{attribute addProperty BoxType "EL5112-0000-0016"}
{attribute addProperty Id "ENC_Status_Channel_1AT %I*ENC_Status_Channel_D7AAABA7128160ENC_Control_Channel_1AT %Q*ENC_Control_Channel_C4E6260B4860WcStateAT %I*WcState_F855686C1620InfoDataAT %I*InfoData_BC63D37F80100"}
{attribute addProperty CRC "1457377746"}
{attribute addProperty SizeInBites "272"}
{attribute addProperty SizeInBytes "34"}
TYPE EL5112_0DC93E84 :
STRUCT
	{attribute addProperty Name "ENC_Status_Channel_1"}
	ENC_Status_Channel_1 : ENC_Status_Channel_D7AAABA7;
	{attribute addProperty Name "ENC_Control_Channel_1"}
	ENC_Control_Channel_1 : ENC_Control_Channel_C4E6260B;
	{attribute addProperty Name "WcState"}
	WcState : WcState_F855686C;
	{attribute addProperty Name "InfoData"}
	InfoData : InfoData_BC63D37F;
END_STRUCT
END_TYPE

(* stored: Version 1.2.0.0, ProductVersion 3.1.4024.9
   DUT EL5112_0DC93E84: Id {13ba9cbc-e8ef-47e0-b007-5b4838b8c32b} *)
